{attribute addProperty BoxType "EL3255-0000-0017"}
{attribute addProperty Id "AI_Standard_ChannelAT %I*ARRAY[0..4] OF AI_Standard_Channel_904746A2160200WcStateAT %I*WcState_98A4DF7520.250InfoDataAT %I*InfoData_BC63D37F80100"}
{attribute addProperty CRC "2682469264"}
{attribute addProperty SizeInBites "242"}
{attribute addProperty SizeInBytes "30.25"}
TYPE EL3255_11D0319B :
STRUCT
	{attribute addProperty Name "AI_Standard_Channel"}
	AI_Standard_Channel : ARRAY[0..4] OF AI_Standard_Channel_904746A2;
	{attribute addProperty Name "WcState"}
	WcState : WcState_98A4DF75;
	{attribute addProperty Name "InfoData"}
	InfoData : InfoData_BC63D37F;
END_STRUCT
END_TYPE

(* stored: Version 1.2.0.0, ProductVersion 3.1.4024.9
   DUT EL3255_11D0319B: Id {3f002ee9-2c6c-4606-8d33-d65cb36dd9a8} *)
